SUBAPPLICATION SwitchPic_5_2 (* Bild umschalten VT und AUX; 5 Zustände *)
  (* Standard: 61499-2 *)
  (* Version 1.0, 2026-05-29, franz *)
  PACKAGE MyLib::sys;
  IMPORT isobus::UT::Q::const::IDs::ID_NULL;
  IMPORT logiBUS::utils::sequence::schieber::SchieberStruct;
  IMPORT logiBUS::utils::sequence::schieber::const::iSTATES::Unknown;
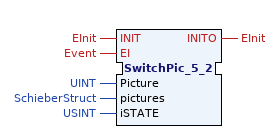
  EVENT_INPUT
    INIT : EInit; (* Initialization Request *)
    EI;
  END_EVENT
  EVENT_OUTPUT
    INITO : EInit; (* Initialization Confirm *)
  END_EVENT
  VAR_INPUT
    Picture : UINT; (* Object ID of the ObjectPointer to the Picture *)
    pictures : logiBUS::utils::sequence::schieber::SchieberStruct := (Unknown := ID_NULL, Closed := ID_NULL, Opening := ID_NULL, Opened := ID_NULL, Closing := ID_NULL); (* the single Pictures *)
    iSTATE : USINT := Unknown;
  END_VAR
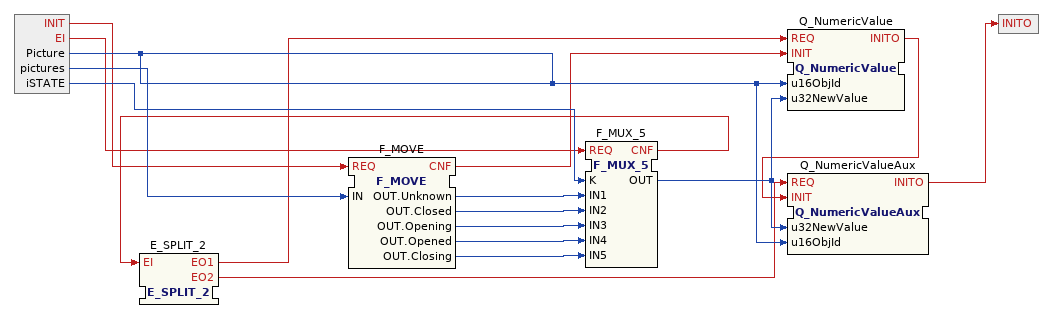
  FBS
    Q_NumericValue : isobus::UT::Q::Q_NumericValue;
    F_MOVE : iec61131::selection::F_MOVE; {SET_ATTRIBUTE(DataType, logiBUS::utils::sequence::schieber::SchieberStruct)}
    F_MUX_5 : iec61131::selection::F_MUX_5;
    Q_NumericValueAux : isobus::UT::Q::Q_NumericValueAux;
    E_SPLIT_2 : iec61499::events::E_SPLIT_2;
  END_FBS
  EVENT_CONNECTIONS
    F_MUX_5.CNF TO E_SPLIT_2.EI;
    E_SPLIT_2.EO1 TO Q_NumericValue.REQ;
    E_SPLIT_2.EO2 TO Q_NumericValueAux.REQ;
    EI TO F_MUX_5.REQ;
    INIT TO F_MOVE.REQ;
    F_MOVE.CNF TO Q_NumericValue.INIT;
    Q_NumericValueAux.INITO TO INITO;
    Q_NumericValue.INITO TO Q_NumericValueAux.INIT;
  END_CONNECTIONS
  DATA_CONNECTIONS
    Picture TO Q_NumericValue.u16ObjId;
    pictures TO F_MOVE.IN;
    iSTATE TO F_MUX_5.K;
    F_MOVE.OUT.Unknown TO F_MUX_5.IN1;
    F_MOVE.OUT.Closed TO F_MUX_5.IN2;
    F_MOVE.OUT.Opening TO F_MUX_5.IN3;
    F_MOVE.OUT.Opened TO F_MUX_5.IN4;
    F_MOVE.OUT.Closing TO F_MUX_5.IN5;
    F_MUX_5.OUT TO Q_NumericValue.u32NewValue;
    F_MUX_5.OUT TO Q_NumericValueAux.u32NewValue;
    Picture TO Q_NumericValueAux.u16ObjId;
  END_CONNECTIONS
END_SUBAPPLICATION
